(*
SPDX-FileCopyrightText: © 2026 Oleksandr Tiutyk <trofimich@gmail.com>
SPDX-License-Identifier: MIT
License: https://opensource.org/license/mit
*)

{attribute 'qualified_only'}
VAR_GLOBAL
	// SA0006: Read-only project namespace string borrowed by tests across tasks.
	{attribute 'analysis' := '-6'}
	Name : STRING := 'TOF_Tests';
END_VAR

(* stored: Version 1.1.0.1, ProductVersion 3.1.4026.13
   GVL CurrentNamespace: Id {5002705f-d70a-4a63-b3f4-fc025d8963f7} *)
